{attribute 'qualified_only'}
{attribute 'strict'}
{attribute 'to_string'}
TYPE EmbarkStationStates :
(
	Init := 0,                                               
	Ready := 1,                                 
	Waiting := 2,
	HasSwitch := 3,
	Call := 4,
	Boarding := 5,
	BoardingComplete := 6,
	Moving := 7,
	ActivateTrackForMover := 8,
	CheckActiveTrack := 9,
	CheckMoverLeft := 10,
	Done := 11,
	test := 20
);
END_TYPE

(* stored: Version 1.1.0.1
   DUT EmbarkStationStates: Id {955ed760-fe4d-452f-958d-eae46f402075} *)
